TEXTLIST TextList_IC6
  0 = 'Rate' | FR: 'Vitesse (Å/s)' | EN: 'Rate (Å/s)'
  1 = 'Thickness' | FR: 'Epaisseur (kÅ)' | EN: 'Thickness (kÅ)'
  2 = 'Détails' | FR: 'Détails...' | EN: 'Details...'
  3 = 'power' | FR: 'Puissance (%)' | EN: 'Power (%)'
  4 = 'Commandes' | FR: ' Commandes' | EN: ' Commands'
  5 = 'start' | FR: 'START' | EN: 'START'
  6 = 'stop' | FR: 'STOP' | EN: 'STOP'
  7 = 'ZERO' | FR: 'ZERO' | EN: 'ZERO'
  8 = 'RESET' | FR: 'RESET' | EN: 'RESET'
  9 = 'etat quartz' | FR: ' Etat des quartz' | EN: ' Crystals state'
  10 = 'fail' | FR: 'FAIL' | EN: 'FAIL'
  11 = 'channel' | FR: 'Canal actif :' | EN: 'Active channel:'
  12 = 'Fréquence' | FR: 'Fréquence' | EN: 'Frequency'
  13 = '% utilisé' | FR: '% utilisé' | EN: 'Life used'
  14 = 'Etat quartz' | FR: 'Etat quartz' | EN: 'Crystal quartz'
   = ''
END_TEXTLIST

(* stored: Version 1.1.0.1, ProductVersion 3.1.4024.10
   TextList TextList_IC6: Id {c7c98635-c504-44f3-9db1-d2bd2dbc0c10} *)
